{attribute 'no_explicit_call' := 'do not call this FB directly'}{attribute 'enable_dynamic_creation'}
FUNCTION_BLOCK FINAL DigitalOutputNode EXTENDS Node
VAR
	output AT %Q* : BOOL;
	in : _BOOL(FALSE);
END_VAR

METHOD PUBLIC Clone : I_Node
VAR
END_VAR
Clone := this^;
END_METHOD

METHOD Dispose
VAR_INPUT
END_VAR
END_METHOD

METHOD FB_init : BOOL
VAR_INPUT
	bInitRetains : BOOL; // if TRUE, the retain variables are initialized (warm start / cold start)
	bInCopyCode : BOOL;  // if TRUE, the instance afterwards gets moved into the copy code (online change)
END_VAR
AddInput('in', in);
END_METHOD

METHOD PROTECTED OnExecute : HRESULT
VAR
END_VAR
output := in.value;
END_METHOD

END_FUNCTION_BLOCK

(* stored: Version 1.1.0.1, ProductVersion 3.1.4024.12
   POU DigitalOutputNode: Id {1a6aa422-dcf5-0618-3bde-508292d00251}, SpecialFunc None
   Folder Constructor: Id {8ccdd20d-570b-0ba5-3267-540f4f9ab370}
   Method Clone: Id {5a10cedc-f20d-00af-1178-3429e0ca0525}
   Method Dispose: Id {e3d041f9-399e-0ad3-1fb7-f682ce1d25fc}
   Method FB_init: Id {55fbf225-9e2c-0c92-2654-70fa2be3a812}
   Method OnExecute: Id {fc8ff28b-a02f-0a31-23a1-6e896590736c} *)
